{attribute 'qualified_only'}
VAR_GLOBAL
	x		: ARRAY [1..4] OF LREAL;
	y		: ARRAY [1..4] OF LREAL; 
	theta	: ARRAY [1..4] OF LREAL;
	
	nPaketlaenge	: UDINT;
	firstByte		: ULINT;
	nextByte		: ULINT;
	sizeLREAL		: ULINT;
END_VAR

(* stored: Version 1.1.0.1, ProductVersion 3.1.4022.3
   GVL UDP: Id {d035a088-9d17-440a-afb8-4ba9d899d630} *)
